FUNCTION_BLOCK FINAL FB_CsvLogger EXTENDS FB_EventLogger  
VAR_INPUT
	Write					: BOOL;							//Write Log
	HeaderString			: ARRAY[0..9] OF STRING;		//Header Strings
	DataString				: ARRAY[0..9] OF STRING;		//Data Strings
END_VAR                                          	    	
VAR_IN_OUT                                          		
	Control					: ST_System;            		//Machine Control Instance
END_VAR                                             		                                           	
VAR                                                     	
	_Export					: BOOL;							//Export CSV to file destination
	_Fault					: BOOL;	     					//Device Fault
	_SeekPos				: DINT;							//Bytes Logged
	_FaultTimer_ET			: REAL;							//Fault timer elapsed
	_fbCreateDir 			: FB_CreateDir;					//Create File Directory Funciton
	_fbFileOpen				: FB_FileOpen;              	//File Open Function      
	_fbFileClose			: FB_FileClose;             	//File Close Function            
    _fbFileRead             : FB_FileRead;              	//File Read Function 			          
    _fbFileWrite            : FB_FileWrite;             	//File Write Function 	          
	_fbFileDelete  			: FB_FileDelete;            	//File Delete Function           
    _fbFileSeek             : FB_FileSeek;              	//File Seek Function             
	_fbFileTell 			: FB_FileTell;              	//File Tell Function 			          
	_fbFindFileEntry 		: FB_EnumFindFileEntry;     	//File Find File Function 		      
    _hSrcFile               : UINT := 0;					//Temporary file handler
 	_hDestFile              : UINT := 0;					//Export file handler
	_Alarm					: BOOL;							//Device Alarm
	_Warning				: BOOL;							//Device Warning
	_AlarmNum				: DINT;							//Device Alarm Number
	_WarningNum				: DINT;							//Device Warning Number
	_ExtendedErrorCode		: UDINT;						//Extended Error Code
	_R_Trig					: ARRAY[0..9] OF R_TRIG;		//Private Rising Edge Triggers
END_VAR
VAR PERSISTENT
	_Enable					: BOOL;							//Enable CSV logging
	_MaxFileSize			: DINT := 100000;           	//Maximum file size in bytes
	_Name					: STRING[15];					//Name for HMI
	_Description			: STRING[40];					//Description for HMI
	_AlarmMute				: BOOL;							//Alarm Mute
	_FaultTimer_PT			: REAL;							//Fault timer preset time
	_TempFilePath			: STRING:='C:\TwinCAT\3.1\Boot\';//Temporary File Path
	_ExportFilePath			: STRING:='C:\TwinCAT\';		//Export File Path
END_VAR

M_AlarmMonitor();
M_WarningMonitor();
M_Log();

{attribute 'monitoring' := 'variable'}
PROPERTY PUBLIC Alarm : Bool
GET
Alarm := _Alarm;
END_GET
END_PROPERTY

{attribute 'monitoring' := 'variable'}
PROPERTY PUBLIC AlarmMute : BOOL
SET
AlarmMute := _AlarmMute;
END_SET
END_PROPERTY

{attribute 'monitoring' := 'variable'}
PROPERTY PUBLIC Description : String[40]
GET
Description := _Description;
END_GET
SET
_Description := Description;
END_SET
END_PROPERTY

{attribute 'monitoring' := 'variable'}
PROPERTY PUBLIC Enable : BOOL
GET
Enable := _Enable;
END_GET
SET
_Enable := Enable;
END_SET
END_PROPERTY

{attribute 'monitoring' := 'variable'}
PROPERTY PUBLIC Fault : Bool
SET
_Fault := Fault;
END_SET
END_PROPERTY

{attribute 'monitoring' := 'variable'}
PROPERTY PUBLIC FaultTimer_ET : real
GET
FaultTimer_ET := _FaultTimer_ET;
END_GET
END_PROPERTY

{attribute 'monitoring' := 'variable'}
PROPERTY PUBLIC FaultTimer_PT : real
GET
FaultTimer_PT := _FaultTimer_PT;
END_GET
SET
_FaultTimer_PT := FaultTimer_PT;
END_SET
END_PROPERTY

METHOD FB_exit : BOOL
VAR_INPUT
	bInCopyCode : BOOL; // if TRUE, the exit method is called for exiting an instance that is copied afterwards (online change).
END_VAR
IF _hSrcFile <> 0 THEN
	_fbFileClose( bExecute := FALSE );	
	_fbFileClose(sNetId:='', hFile:=_hSrcFile, bExecute:=TRUE, tTimeout:=DEFAULT_ADS_TIMEOUT);
END_IF
END_METHOD

METHOD PRIVATE M_AlarmMonitor
VAR_INPUT
END_VAR
VAR_INST // added by the converter: edge detectors and wires of the graphical bodies
    _w1, _w2, _w3, _w4, _w5, _w6, _w7 : BOOL;
    _rt1, _rt2, _rt3, _rt4, _rt5, _rt6, _rt7, _rt8, _rt9, _rt10 : R_TRIG;
END_VAR
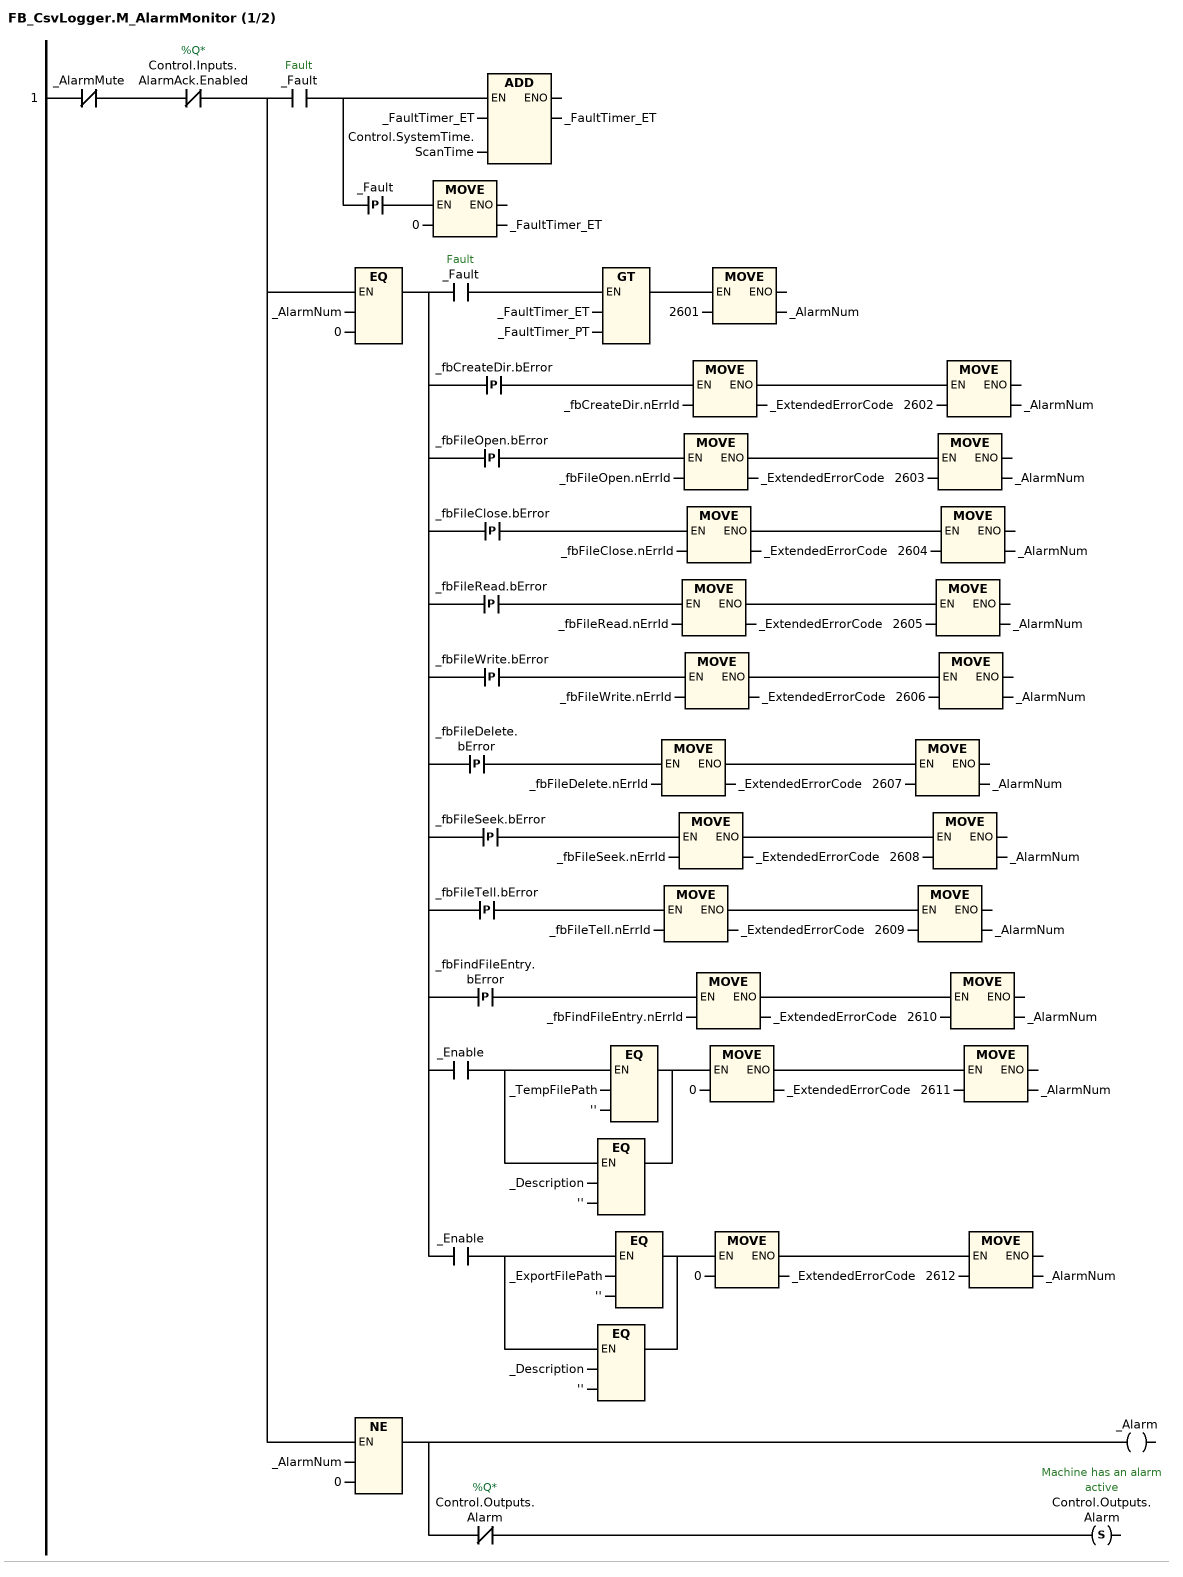
// NETWORK 1
//   Control.Inputs.AlarmAck.Enabled: AT %Q*
//   _Fault: Fault
//   _FaultTimer_ET: Fault timer elapsed
//   Control.SystemTime.ScanTime: Last scan time (Seconds)
//   _FaultTimer_PT: Fault timer preset time
//   Control.Outputs.Alarm: AT %Q* | Machine has an alarm active
_w1 := NOT _AlarmMute AND NOT Control.Inputs.AlarmAck.Enabled;
_w2 := _w1 AND _Fault;
IF _w2 THEN _FaultTimer_ET := _FaultTimer_ET + Control.SystemTime.ScanTime; END_IF
_rt1(CLK := _Fault);
IF _w2 AND _rt1.Q THEN _FaultTimer_ET := 0; END_IF
_w3 := _w1 AND _AlarmNum = 0;
IF _w3 AND _Fault AND _FaultTimer_ET > _FaultTimer_PT THEN _AlarmNum := 2601; END_IF
_rt2(CLK := _fbCreateDir.bError);
IF _w3 AND _rt2.Q THEN _ExtendedErrorCode := _fbCreateDir.nErrId; END_IF
IF _w3 AND _rt2.Q THEN _AlarmNum := 2602; END_IF
_rt3(CLK := _fbFileOpen.bError);
IF _w3 AND _rt3.Q THEN _ExtendedErrorCode := _fbFileOpen.nErrId; END_IF
IF _w3 AND _rt3.Q THEN _AlarmNum := 2603; END_IF
_rt4(CLK := _fbFileClose.bError);
IF _w3 AND _rt4.Q THEN _ExtendedErrorCode := _fbFileClose.nErrId; END_IF
IF _w3 AND _rt4.Q THEN _AlarmNum := 2604; END_IF
_rt5(CLK := _fbFileRead.bError);
IF _w3 AND _rt5.Q THEN _ExtendedErrorCode := _fbFileRead.nErrId; END_IF
IF _w3 AND _rt5.Q THEN _AlarmNum := 2605; END_IF
_rt6(CLK := _fbFileWrite.bError);
IF _w3 AND _rt6.Q THEN _ExtendedErrorCode := _fbFileWrite.nErrId; END_IF
IF _w3 AND _rt6.Q THEN _AlarmNum := 2606; END_IF
_rt7(CLK := _fbFileDelete.bError);
IF _w3 AND _rt7.Q THEN _ExtendedErrorCode := _fbFileDelete.nErrId; END_IF
IF _w3 AND _rt7.Q THEN _AlarmNum := 2607; END_IF
_rt8(CLK := _fbFileSeek.bError);
IF _w3 AND _rt8.Q THEN _ExtendedErrorCode := _fbFileSeek.nErrId; END_IF
IF _w3 AND _rt8.Q THEN _AlarmNum := 2608; END_IF
_rt9(CLK := _fbFileTell.bError);
IF _w3 AND _rt9.Q THEN _ExtendedErrorCode := _fbFileTell.nErrId; END_IF
IF _w3 AND _rt9.Q THEN _AlarmNum := 2609; END_IF
_rt10(CLK := _fbFindFileEntry.bError);
IF _w3 AND _rt10.Q THEN _ExtendedErrorCode := _fbFindFileEntry.nErrId; END_IF
IF _w3 AND _rt10.Q THEN _AlarmNum := 2610; END_IF
_w4 := _w3 AND _Enable;
IF _w4 AND _TempFilePath = '' OR _w4 AND _Description = '' THEN _ExtendedErrorCode := 0; END_IF
IF _w4 AND _TempFilePath = '' OR _w4 AND _Description = '' THEN _AlarmNum := 2611; END_IF
_w5 := _w3 AND _Enable;
IF _w5 AND _ExportFilePath = '' OR _w5 AND _Description = '' THEN _ExtendedErrorCode := 0; END_IF
IF _w5 AND _ExportFilePath = '' OR _w5 AND _Description = '' THEN _AlarmNum := 2612; END_IF
_w6 := _w1 AND _AlarmNum <> 0;
_Alarm := _w6;
Control.Outputs.Alarm S= _w6 AND NOT Control.Outputs.Alarm;

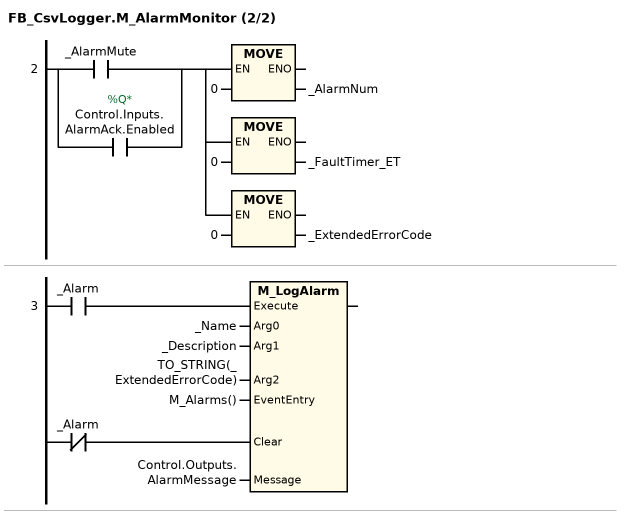
// NETWORK 2
//   Control.Inputs.AlarmAck.Enabled: AT %Q*
//   _FaultTimer_ET: Fault timer elapsed
//   _ExtendedErrorCode: Fault timer elapsed
_w7 := _AlarmMute OR Control.Inputs.AlarmAck.Enabled;
IF _w7 THEN _AlarmNum := 0; END_IF
IF _w7 THEN _FaultTimer_ET := 0; END_IF
IF _w7 THEN _ExtendedErrorCode := 0; END_IF

// NETWORK 3
M_LogAlarm(Execute := _Alarm, Arg0 := _Name, Arg1 := _Description, Arg2 := TO_STRING(_ExtendedErrorCode), EventEntry := M_Alarms(), Clear := NOT _Alarm, Message := Control.Outputs.AlarmMessage);
END_METHOD

METHOD PRIVATE M_Alarms : TcEventEntry
VAR_INPUT
END_VAR
CASE _AlarmNum OF
	2601: M_Alarms:= TC_Events.TcCsvLogger.A_2601;//Alarm
	2602: M_Alarms:= TC_Events.TcCsvLogger.A_2602;//Create File Directory Error 
	2603: M_Alarms:= TC_Events.TcCsvLogger.A_2603;//File Open Error
	2604: M_Alarms:= TC_Events.TcCsvLogger.A_2604;//File Close Error
	2605: M_Alarms:= TC_Events.TcCsvLogger.A_2605;//File Read Error			
	2606: M_Alarms:= TC_Events.TcCsvLogger.A_2606;//File Write Error		
	2607: M_Alarms:= TC_Events.TcCsvLogger.A_2607;//File Delete Error	
	2608: M_Alarms:= TC_Events.TcCsvLogger.A_2608;//File Seek Error
	2609: M_Alarms:= TC_Events.TcCsvLogger.A_2609;//File Tell Error			
	2610: M_Alarms:= TC_Events.TcCsvLogger.A_2610;//File Find File Error		
	2611: M_Alarms:= TC_Events.TcCsvLogger.A_2611;//Temporary File Path or Name Error		
	2612: M_Alarms:= TC_Events.TcCsvLogger.A_2612;//Export File Path or Name Error				
ELSE
	M_Alarms:= TC_Events.TcCsvLogger.A_Undefined;
END_CASE
END_METHOD

METHOD PUBLIC M_Log
VAR_INST
	{attribute 'tc_no_symbol'}
	_Step								: UINT;
	{attribute 'tc_no_symbol'}
	_Timeout							: TON;
	{attribute 'tc_no_symbol'}
    _buffRead                			: ARRAY[1..100000] OF BYTE;
	{attribute 'tc_no_symbol'}
 	_cbReadLength            			: UDINT := 0;
	{attribute 'tc_no_symbol'}
	_HeaderString						: T_MAXSTRING;
	{attribute 'tc_no_symbol'}
	_DataString							: T_MAXSTRING;
	{attribute 'tc_no_symbol'}
	_TimeStamp							: STRING(31);
	{attribute 'tc_no_symbol'}
	_Value								: INT;
END_VAR
CASE _Step OF
	0:  // Step 0: Wait for open file request
		IF _Enable AND NOT _Alarm THEN
			_Step := 1; 
		END_IF
	1:  // Step 1: Check if temporary directory exists	
		_fbFindFileEntry(bExecute:= FALSE);
		_fbFindFileEntry(sPathName:= LEFT(_TempFilePath,LEN(_TempFilePath)-1), eCmd:= eEnumCmd_First, bExecute:= TRUE, tTimeout:= DEFAULT_ADS_TIMEOUT);
		IF _fbFindFileEntry.bBusy THEN _Step := 2; END_IF
	2:  // Step 2: Wait for temporary directory check	
		_fbFindFileEntry( bExecute := FALSE );
		IF NOT _fbFindFileEntry.bBusy AND NOT _fbFindFileEntry.bError THEN 
			IF _fbFindFileEntry.stFindFile.fileAttributes.bDirectory THEN
				_Step := 5; 
			ELSE
				_Step := 3; 
			END_IF
		END_IF
	3:  // Step 3: Create temporary directory
	    _hSrcFile:=0;
		_fbCreateDir( bExecute := FALSE );
		_fbCreateDir(sNetId:= '', sPathName := _TempFilePath, ePath:= PATH_GENERIC, bExecute:= TRUE, tTimeout:= DEFAULT_ADS_TIMEOUT);
		IF _fbCreateDir.bBusy THEN _Step := 4; END_IF
	4:  // Step 4: Wait for temporary directory to be created
		_fbCreateDir( bExecute := FALSE );
		IF NOT _fbCreateDir.bBusy AND NOT _fbCreateDir.bError THEN _Step := 5; END_IF
	5:  // Step 5: Check if temporary file exists	
		_fbFindFileEntry(bExecute:= FALSE);
		_fbFindFileEntry(sPathName:= concat(_TempFilePath,concat(_Description,'.csv')), eCmd:= eEnumCmd_First, bExecute:= TRUE, tTimeout:= DEFAULT_ADS_TIMEOUT);
		IF _fbFindFileEntry.bBusy THEN _Step := 6; END_IF
	6:  // Step 6: Wait for temporary file check	
		_fbFindFileEntry( bExecute := FALSE );
		IF NOT _fbFindFileEntry.bBusy AND NOT _fbFindFileEntry.bError THEN 
			IF _fbFindFileEntry.stFindFile.fileAttributes.bArchive THEN
				_fbFileOpen.nMode := FOPEN_MODEREAD OR FOPEN_MODEPLUS;
			ELSE
				_fbFileOpen.nMode := FOPEN_MODEWRITE; 
			END_IF
			_Step := 7; 
		END_IF	
	7:  // Step 7: Open temporary CSV file
		_fbFileOpen( bExecute := FALSE );
		_fbFileOpen( sNetId := '', sPathName := concat(_TempFilePath,concat(_Description,'.csv')), ePath := PATH_GENERIC, tTimeout := DEFAULT_ADS_TIMEOUT, bExecute := TRUE );
		IF _fbFileOpen.bBusy THEN _Step := 8; END_IF
	8:	// Step 8: Wait for temporary CSV to be created
		_fbFileOpen( bExecute := FALSE, hFile=> _hSrcFile);
		IF NOT _fbFileOpen.bBusy AND NOT _fbFileOpen.bError THEN 
			IF _fbFileOpen.nMode = (FOPEN_MODEREAD OR FOPEN_MODEPLUS) THEN
				_Step := 9; 
			ELSE
				_Step := 11; 
			END_IF
		END_IF	
	9:  // Step 9: Find if header exists 
        _fbFileRead( bExecute:= FALSE );
        _fbFileRead( sNetId:='', hFile:=_hSrcFile, bExecute:=TRUE, pReadBuff:= ADR(_buffRead), cbReadLen:= SIZEOF(_buffRead), tTimeout:=DEFAULT_ADS_TIMEOUT);
        _Step := 10;
    10:  // Step 10: Wait for feedback of header existance
        _fbFileRead( bExecute:= FALSE );
        IF NOT _fbFileRead.bBusy AND NOT _fbFileRead.bError THEN
			IF _fbFileRead.cbReadLen > 0 THEN // Header already exists
				_Step := 13; 
			ELSE
				_Step := 11; 
			END_IF
        END_IF
	11:	// Step 11: Write header string to temporary CSV file
		_fbFileWrite( bExecute := FALSE);
		_HeaderString := '';
		FOR _Value:= 0 TO UINT_TO_INT(SIZEOF(HeaderString)/SIZEOF(STRING))-1 BY 1 DO
			IF _Value < UINT_TO_INT((SIZEOF(HeaderString)/SIZEOF(STRING))-1) THEN
				IF HeaderString[_Value+1] <> '' THEN
			    	_HeaderString := concat(_HeaderString,concat(HeaderString[_Value],','));	
				ELSE
					_HeaderString := concat(_HeaderString,concat(HeaderString[_Value],'$0D'));
					EXIT;
				END_IF
			ELSE
				_HeaderString := concat(_HeaderString,concat(HeaderString[_Value],'$0D'));
			END_IF 
		END_FOR;
		_fbFileWrite( sNetId:='', hFile:= _hSrcFile, pWriteBuff:= ADR(_HeaderString), cbWriteLen:= INT_TO_UINT(Len(_HeaderString)), bExecute:=TRUE, tTimeout:=DEFAULT_ADS_TIMEOUT);
		IF _fbFileWrite.bBusy THEN _Step := 12; END_IF
	12:	// Step 12: Wait for CSV header to be written
		_fbFileWrite( bExecute := FALSE );
		IF NOT _fbFileWrite.bBusy AND NOT _fbFileWrite.bError THEN 
			_Step := 13; 
		END_IF	
	13:	// Step 13: Get the current position of the file pointer
		_fbFileTell(bExecute:= FALSE);
		_fbFileTell(hFile:= _hSrcFile, bExecute:= TRUE);
		IF _fbFileTell.bBusy THEN _Step := 14; END_IF
	14:	// Step 14: Wait for file tell
		_fbFileTell(bExecute:= FALSE, nSeekPos => _SeekPos);
		IF NOT _fbFileTell.bBusy AND NOT _fbFileTell.bError THEN 
			_Step := 15; 
		END_IF	
	15:	// Step 15: Set the current position of the file pointer
		_fbFileSeek(bExecute:= FALSE);
		_fbFileSeek(eOrigin:= SEEK_SET, nSeekPos:= _SeekPos + 1, hFile:= _hSrcFile, bExecute:= TRUE);
		IF _fbFileSeek.bBusy THEN _Step := 16; END_IF
	16:	// Step 16: Wait for file seek
		_fbFileSeek(bExecute:= FALSE);
		IF NOT _fbFileSeek.bBusy AND NOT _fbFileSeek.bError THEN 
			_Step := 17; 
		END_IF	
	17: // Step 17: Wait for write or export request
		_R_Trig[0](CLK:= _Export);
		_R_Trig[1](CLK:= Write);
		IF _R_Trig[0].Q THEN
			_Step := 22;
		ELSIF _R_Trig[1].Q THEN
 			_Step := 18;
		ELSIF NOT _Enable THEN
			_Step := 36;
		END_IF
	18:	// Step 18: Write data to CSV file
		_fbFileWrite( bExecute := FALSE);
		_DataString := '';
		FOR _Value:= 0 TO UINT_TO_INT(SIZEOF(DataString)/SIZEOF(STRING))-1 BY 1 DO
			IF _Value < UINT_TO_INT((SIZEOF(DataString)/SIZEOF(STRING))-1) THEN
				IF DataString[_Value+1] <> '' THEN
			    	_DataString := concat(_DataString,concat(DataString[_Value],','));	
				ELSE
					_DataString := concat(_DataString,concat(DataString[_Value],'$0D'));
					EXIT;
				END_IF
			ELSE
				_DataString := concat(_DataString,concat(DataString[_Value],'$0D'));
			END_IF 
		END_FOR;
		_fbFileWrite( sNetId:='', hFile:= _hSrcFile, pWriteBuff:= ADR(_DataString), cbWriteLen:= INT_TO_UINT(Len(_DataString)), bExecute:=TRUE, tTimeout:=T#3S );
		IF _fbFileWrite.bBusy THEN _Step := 19; END_IF
	19:	// Step 19: Wait for CSV data to be written
		_fbFileWrite( bExecute := FALSE );
		IF NOT _fbFileWrite.bBusy AND NOT _fbFileWrite.bError THEN 
			_Step := 20; 
		END_IF		
	20:	// Step 20: Get the current position of the file pointer
		_fbFileTell(bExecute:= FALSE);
		_fbFileTell(hFile:= _hSrcFile, bExecute:= TRUE);
		IF _fbFileTell.bBusy THEN _Step := 21; END_IF
	21:	// Step 21: Wait for file tell
		_fbFileTell(bExecute:= FALSE, nSeekPos => _SeekPos);
		IF NOT _fbFileTell.bBusy AND NOT _fbFileTell.bError THEN 
			IF (_SeekPos > _MaxFileSize) OR (DINT_TO_UDINT(_SeekPos) > SIZEOF(_buffRead)) THEN
				_SeekPos := LEN(_HeaderString);
				_Step := 15; 
			ELSE 
				_Step := 17; 
			END_IF
		END_IF	
	22: // Step 22: Close temporary CSV 
		IF _hSrcFile <> 0 THEN
			_fbFileClose( bExecute := FALSE );	
			_fbFileClose(sNetId:='', hFile:=_hSrcFile, bExecute:=TRUE, tTimeout:=DEFAULT_ADS_TIMEOUT);
			IF _fbFileClose.bBusy THEN _Step := 23; END_IF
		ELSE
			_Step := 24;
		END_IF
	23:	// Step 23: Wait for temporary CSV to close
		_fbFileClose( bExecute := FALSE );
		IF NOT _fbFileClose.bBusy AND NOT _fbFileClose.bError THEN 
			_hSrcFile := 0;
			_Step := 24;
		END_IF
	24: // Step 24: Open temporary CSV file
		_fbFileOpen( bExecute := FALSE );
		_fbFileOpen( sNetId := '', sPathName := concat(_TempFilePath,concat(_Description,'.csv')),nMode := FOPEN_MODEREAD, ePath := PATH_GENERIC, tTimeout := DEFAULT_ADS_TIMEOUT, bExecute := TRUE );
		IF _fbFileOpen.bBusy THEN _Step := 25; END_IF
	25:	// Step 25: Wait for temporary CSV to be created
		_fbFileOpen( bExecute := FALSE, hFile=> _hSrcFile);
		IF NOT _fbFileOpen.bBusy AND NOT _fbFileOpen.bError THEN _Step := 26; END_IF	
	26: // Step 26: Check if export directory exists	
		_fbFindFileEntry(bExecute:= FALSE);
		_fbFindFileEntry(sPathName:= LEFT(_ExportFilePath,LEN(_ExportFilePath)-1), eCmd:= eEnumCmd_First, bExecute:= TRUE, tTimeout:= DEFAULT_ADS_TIMEOUT);
		IF _fbFindFileEntry.bBusy THEN _Step := 27; END_IF
	27: // Step 27: Wait for export directory check	
		_fbFindFileEntry( bExecute := FALSE );
		IF NOT _fbFindFileEntry.bBusy AND NOT _fbFindFileEntry.bError THEN 
			IF _fbFindFileEntry.stFindFile.fileAttributes.bDirectory THEN
				_Step := 30; 
			ELSE
				_Step := 28; 
			END_IF
		END_IF
	28: // Step 28: Create export directory
        _hDestFile:=0;
		_fbCreateDir( bExecute := FALSE );
		_fbCreateDir(sNetId:= '', sPathName := _ExportFilePath, ePath:= PATH_GENERIC, bExecute:= TRUE, tTimeout:= DEFAULT_ADS_TIMEOUT);
		IF _fbCreateDir.bBusy AND NOT _fbCreateDir.bError THEN _Step := 29; END_IF
	29: // Step 29: Wait for export directory to be created
		_fbCreateDir( bExecute := FALSE );
		IF NOT _fbCreateDir.bBusy THEN _Step := 30; END_IF
	30: // Step 30: Create export CSV file
		_fbFileOpen( bExecute := FALSE );
		_timeStamp := concat(LEFT(SystemTime_To_String(Control.SystemTime.CurrentTime),10),concat(' ',concat(TO_STRING(Control.SystemTime.CurrentTime.wHour),concat('-',concat(TO_STRING(Control.SystemTime.CurrentTime.wMinute),concat('-',TO_STRING(Control.SystemTime.CurrentTime.wSecond)))))));
		_fbFileOpen( sNetId := '', sPathName := concat(_ExportFilePath,concat(_TimeStamp,concat(' ',concat(_Description,'.csv')))),nMode := FOPEN_MODEAPPEND, ePath := PATH_GENERIC, tTimeout := DEFAULT_ADS_TIMEOUT, bExecute := TRUE );
		IF _fbFileOpen.bBusy THEN _Step := 31; END_IF
	31:	// Step 31: Wait for export CSV to be created
		_fbFileOpen( bExecute := FALSE, hFile=> _hDestFile);
		IF NOT _fbFileOpen.bBusy AND NOT _fbFileOpen.bError THEN _Step := 32; END_IF	
    32: // Step 32: Read data from temporary file 
        _cbReadLength := 0;
        _fbFileRead( bExecute:= FALSE );
        _fbFileRead( sNetId:='', hFile:=_hSrcFile , pReadBuff:= ADR(_buffRead), cbReadLen:= SIZEOF(_buffRead),bExecute:=TRUE, tTimeout:=T#60S);
        _Step := 33;
    33:	// Step 33: Wait for temporary file to be read
        _fbFileRead( bExecute:= FALSE );
        IF NOT _fbFileRead.bBusy AND NOT _fbFileRead.bError THEN
        	_cbReadLength := _fbFileRead.cbRead;
            _Step := 34;
        END_IF
    34: // Step 34: Write data to export file 
        _fbFileWrite( bExecute := FALSE );
        _fbFileWrite( sNetId:='', hFile:=_hDestFile,pWriteBuff:= ADR(_buffRead), cbWriteLen:= _cbReadLength, bExecute:=TRUE, tTimeout:=T#60S);
        _Step := 35;
    35: // Step 35: Wait for export file to be written
       	_fbFileWrite( bExecute := FALSE );
        IF NOT _fbFileWrite.bBusy THEN
             IF _fbFileWrite.bError THEN
                  _Step := 42;
             ELSE
             	IF _fbFileRead.bEOF THEN//Check if the EOF flag ist set 
                   _Step := 36;//Cleanup: close the export and temporary files 
               	ELSE
                   _Step := 32;//Repeat reading/writing 
               	END_IF
            END_IF
        END_IF
	36: // Step 36: Close export CSV file
		IF _hDestFile <> 0 THEN
			_fbFileClose( bExecute := FALSE );	
			_fbFileClose(sNetId:='', hFile:=_hDestFile, bExecute:=TRUE, tTimeout:=DEFAULT_ADS_TIMEOUT);
			IF _fbFileClose.bBusy THEN _Step := 37; END_IF
		ELSE
			_Step := 38;
		END_IF
	37:	// Step 37: Wait for export CSV to close
		_fbFileClose( bExecute := FALSE );
		IF NOT _fbFileClose.bBusy AND NOT _fbFileClose.bError THEN 
			_hDestFile := 0;
			_Step := 38;
		END_IF
	38: // Step 38: Close temporary CSV file
		IF _hSrcFile <> 0 THEN
			_fbFileClose( bExecute := FALSE );	
			_fbFileClose(sNetId:='', hFile:=_hSrcFile, bExecute:=TRUE, tTimeout:=DEFAULT_ADS_TIMEOUT);
			IF _fbFileClose.bBusy THEN _Step := 39; END_IF
		ELSE
			_Step := 42;
		END_IF
	39:	// Step 39: Wait for temporary CSV to close
		_fbFileClose( bExecute := FALSE );
		IF NOT _fbFileClose.bBusy AND NOT _fbFileClose.bError THEN 
			_hSrcFile := 0;
			_Step := 40;
		END_IF
	40:  // Step 40: Delete temporary CSV file
		_fbFileDelete( bExecute := FALSE );	
		_fbFileDelete(sNetId:='', sPathName:= concat(_TempFilePath,concat(_Description,'.csv')), ePath:= PATH_GENERIC, bExecute:=TRUE, tTimeout:=DEFAULT_ADS_TIMEOUT);
		IF _fbFileDelete.bBusy THEN _Step := 41; END_IF
	41:	// Step 33: Wait for temporary CSV to Delete
		_fbFileDelete( bExecute := FALSE );
		IF NOT _fbFileDelete.bBusy AND NOT _fbFileDelete.bError THEN 
			_Step := 42;
		END_IF
    42: // Step 42: Cleanup 
        IF _hDestFile <> 0 THEN
        	_Step := 36;//Close the export file
        ELSIF _hSrcFile <> 0 THEN
        	_Step := 38;//Close and delete the temporary file 
        ELSE
        	_Step := 0;
        END_IF	
	
END_CASE

// Error Handling
_Timeout(In:=_Step > 0 AND _Step <> 17 ,PT:=T#60S);
_R_Trig[6](clk:= _Timeout.Q OR _Alarm);
IF _R_Trig[6].Q THEN _STEP := 36; END_IF
END_METHOD

METHOD PRIVATE M_WarningMonitor
VAR_INPUT
END_VAR
VAR_INST
END_VAR
VAR_INST // added by the converter: edge detectors and wires of the graphical bodies
    _w1 : BOOL;
END_VAR
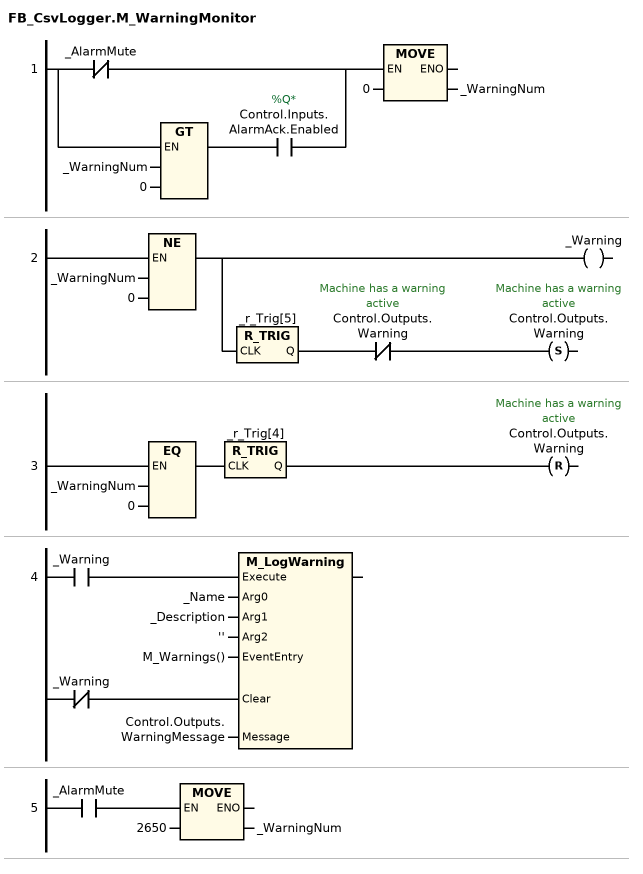
// NETWORK 1
//   Control.Inputs.AlarmAck.Enabled: AT %Q*
IF NOT _AlarmMute OR _WarningNum > 0 AND Control.Inputs.AlarmAck.Enabled THEN _WarningNum := 0; END_IF

// NETWORK 2
//   Control.Outputs.Warning: Machine has a warning active
_w1 := _WarningNum <> 0;
_Warning := _w1;
_r_Trig[5](CLK := _w1); // R_TRIG
Control.Outputs.Warning S= _r_Trig[5].Q AND NOT Control.Outputs.Warning;

// NETWORK 3
//   Control.Outputs.Warning: Machine has a warning active
_r_Trig[4](CLK := _WarningNum = 0); // R_TRIG
Control.Outputs.Warning R= _r_Trig[4].Q;

// NETWORK 4
M_LogWarning(Execute := _Warning, Arg0 := _Name, Arg1 := _Description, Arg2 := '', EventEntry := M_Warnings(), Clear := NOT _Warning, Message := Control.Outputs.WarningMessage);

// NETWORK 5
IF _AlarmMute THEN _WarningNum := 2650; END_IF
END_METHOD

METHOD PRIVATE M_Warnings : TcEventEntry
VAR_INPUT
END_VAR
CASE _WarningNum OF
	2650: M_Warnings:= TC_Events.TcCsvLogger.W_2650;//Alarm Mute							
ELSE
	M_Warnings:=  TC_Events.TcCsvLogger.W_Undefined;
END_CASE
END_METHOD

{attribute 'monitoring' := 'variable'}
PROPERTY PUBLIC Name : String[15]
GET
Name := _Name;
END_GET
SET
_Name := Name;
END_SET
END_PROPERTY

{attribute 'monitoring' := 'variable'}
PROPERTY PUBLIC Warning : Bool
GET
Warning := _Warning;
END_GET
END_PROPERTY

END_FUNCTION_BLOCK

(* stored: Version 1.1.0.1, ProductVersion 3.1.4024.3
   POU FB_CsvLogger: Id {c2537169-58c7-4370-97f6-0daeb6e4d0fc}, SpecialFunc None
   Property Alarm: Id {16417da4-486e-4c76-8e7f-d195ecdf03e7}
   Get Get: Id {abf8e61f-aaf0-413a-9a91-b8caea2d7352}
   Property AlarmMute: Id {57950896-07e9-4c83-9916-32932200c508}
   Set Set: Id {61f7b05a-024b-4138-82b7-91a72d0c0cb2}
   Property Description: Id {8595a6a9-874d-4ee1-8cd2-e265bce4ab47}
   Get Get: Id {e4b6ff03-0122-48c6-9e59-b0c9c0c6a429}
   Set Set: Id {fbe918fe-537e-4a9e-b6af-91efa72a2352}
   Property Enable: Id {c8039498-9c84-4127-b3fc-ed15eabb15e0}
   Get Get: Id {22800e69-029f-4c98-8d29-28811c1af04f}
   Set Set: Id {35533289-1301-4e53-84f3-a41299ebf337}
   Property Fault: Id {5ed0e534-d409-4786-8d4e-5240817d8fca}
   Set Set: Id {005d4830-f29f-4986-b036-2934dbdc3a35}
   Property FaultTimer_ET: Id {d9bdcb8f-7999-442a-818e-a92c2b891455}
   Get Get: Id {90c48135-8309-4fe2-874e-5f656d054389}
   Property FaultTimer_PT: Id {23fdaf2d-3a10-45f6-a232-f23999e44f6d}
   Get Get: Id {defcb7a5-affc-4adc-8ca6-4b621ec3500e}
   Set Set: Id {b2d8a789-e1a1-4f1d-8b78-bdaf5ffc3fd6}
   Method FB_exit: Id {3320c26a-743b-434a-a643-7c17f86126ae}
   Method M_AlarmMonitor: Id {74e5e18b-528d-42ca-a325-3ba534e6ce7f}
   Method M_Alarms: Id {a428ca24-c463-4247-b85e-f51252b43597}
   Method M_Log: Id {95ac5f65-29f3-4d1d-8d05-724606148416}
   Method M_WarningMonitor: Id {30e564e5-1b8b-42c6-a8de-fbe9a806a35b}
   Method M_Warnings: Id {1933252e-cae6-45a4-a875-1e9a9a5afd6a}
   Property Name: Id {82876ba0-425b-4d50-8705-5d30278e4822}
   Get Get: Id {7d7c9ece-e123-409f-853a-9aeb2e0d8941}
   Set Set: Id {561edddf-3182-4bb5-a0df-a90c5c3abc2d}
   Property Warning: Id {1f851916-63b2-4483-aa1a-e7cdd5c1405c}
   Get Get: Id {c0701230-83e8-4c2a-86b1-c1f5d2915242} *)
